// TIA Portal V20 export
TYPE "zd_SCS_ModeBox_InOut"
// stored: Access Published, IsFailsafeCompliant true, Namespace Safety
   STRUCT
      SCSInput : "Safety.zd_SCS_ModeBox_Inputs";
      FaultReset : Bool;
      GuardsOK : Bool;
      SCSFaulted : Bool;
      SCSAckReq : Bool;
      CellAuto : Bool;
      AllMotionOFF : Bool;
      SCSOutputs : "Safety.zd_SCS_ModeBox_Outputs";
      SCSOutputsLT : "Safety.zd_SCS_ModeBox_OutputsLT";
      HazardsRemoved { S7_SetPoint := 'True'} : Bool;
      PendantReqHazControl : Bool;
      Faulted : Bool;
      AckReq : Bool;
   END_STRUCT;
END_TYPE
